// TwinCAT 3 PLC project Tc3EventLoggerUsage
// ProgramVersion: 3.1.4022.0
// libraries:
//   Tc2_MC2, * (Beckhoff Automation GmbH)
//   Tc2_Standard, * (Beckhoff Automation GmbH)
//   Tc2_System, * (Beckhoff Automation GmbH)
//   Tc2_Utilities, * (Beckhoff Automation GmbH)
//   Tc3_EventLogger, * (Beckhoff Automation GmbH)
//   Tc3_Module, * (Beckhoff Automation GmbH)
// project tree:
//   / GlobalTextList.TcGTLO, PlcTask.TcTTO, Visualization Manager.TcVMO (not stored), VISU_TASK.TcTTO
//   POUs/ FB_CONTROL.TcPOU, MAIN.TcPOU
//   VISUs/ Visualization.TcVIS
// (motion and I/O tree: see PLC project adslogeventexample)
// real-time tasks:
//   TASK PlcTask: cycle T#10ms, priority 20, ADS port 350
//   TASK VISU_TASK: cycle T#200000us, priority 30, ADS port 351
// variable links:
//   Tc3EventLoggerUsage/Tc3EventLoggerUsage Instance <-> NC-Task 1 SAF/Axes/Axis 1
//     PlcTask Inputs/MAIN.Axis.NcToPlc <-> Outputs/ToPlc
//     PlcTask Outputs/MAIN.Axis.PlcToNc <-> Inputs/FromPlc

CONFIGURATION Tc3EventLoggerUsage
    RESOURCE PLC ON TwinCAT3
        TASK PlcTask(INTERVAL := T#10ms, PRIORITY := 20);
        TASK VISU_TASK(INTERVAL := T#200000us, PRIORITY := 30);
        PROGRAM MAIN WITH PlcTask : MAIN;
        PROGRAM VisuElems_Visu_Prg WITH VISU_TASK : VisuElems.Visu_Prg;
    END_RESOURCE
END_CONFIGURATION

// ---- POUs/MAIN.TcPOU
PROGRAM MAIN
VAR
	control:fb_control;
	ServoPower:MC_Power;
	ServoReset:MC_Reset;
	Axis: AXIS_REF;
	Events:FB_AdsReadEvents;
	nNumberOfEvents: UDINT;
	bBusy: BOOL;
	bDone: BOOL;
	bError: BOOL;
	nErrId: UDINT;
END_VAR

control(Start:= control.Start, McOutputs=> , Axis:= Axis);

ServoPower(
	Axis:= Axis, 
	Enable:= ServoPower.Enable, 
	Enable_Positive:= TRUE, 
	Enable_Negative:= TRUE, 
	Override:= , 
	BufferMode:= MC_Aborting, 
	Options:= , 
	Status=> , 
	Busy=> , 
	Active=> , 
	Error=> , 
	ErrorID=> );

ServoReset(
	Axis:= Axis, 
	Execute:= ServoReset.Execute, 
	Done=> , 
	Busy=> , 
	Error=> , 
	ErrorID=> );	

	
Events(
	sNetId:= '', 
	bReadEvents:= Events.bReadEvents, 
	nLanguageId:= 1033, 
	eDateAndTimeFormat:= E_DateAndTimeFormat.de_DE, 
	tRefreshTime:= T#1S, 
	tTimeout:= T#5S, 
	aEvents=> , 
	nNumberOfEvents=> nNumberOfEvents, 
	bBusy=> bBusy, 
	bDone=> bDone, 
	bError=> bError, 
	nErrId=> nErrId);

END_PROGRAM

// ---- POUs/FB_CONTROL.TcPOU
FUNCTION_BLOCK FB_CONTROL
VAR_INPUT
	Start:BOOL;
END_VAR
VAR_OUTPUT
	McOutputs:ST_McOutputs;
END_VAR
VAR
	MoveAbsolute:MC_MoveAbsolute;
END_VAR

VAR_IN_OUT
	Axis: AXIS_REF;
END_VAR

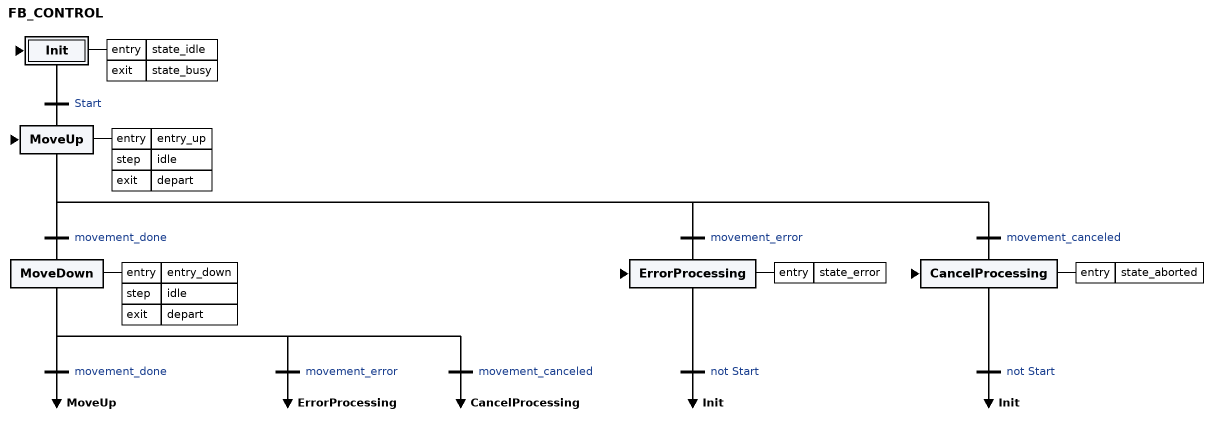
INITIAL_STEP Init:
    state_idle(P1);  // entry action
    state_busy(P0);  // exit action
END_STEP
TRANSITION FROM Init TO MoveUp
    := Start;
END_TRANSITION
STEP MoveUp:
    entry_up(P1);  // entry action
    idle(N);  // step action
    depart(P0);  // exit action
END_STEP
TRANSITION FROM MoveUp TO MoveDown
    := movement_done;
END_TRANSITION
TRANSITION FROM MoveUp TO ErrorProcessing
    := movement_error;
END_TRANSITION
STEP ErrorProcessing:
    state_error(P1);  // entry action
END_STEP
TRANSITION FROM ErrorProcessing TO Init
    := not Start;
END_TRANSITION
TRANSITION FROM MoveUp TO CancelProcessing
    := movement_canceled;
END_TRANSITION
STEP CancelProcessing:
    state_aborted(P1);  // entry action
END_STEP
TRANSITION FROM CancelProcessing TO Init
    := not Start;
END_TRANSITION
STEP MoveDown:
    entry_down(P1);  // entry action
    idle(N);  // step action
    depart(P0);  // exit action
END_STEP
TRANSITION FROM MoveDown TO MoveUp
    := movement_done;
END_TRANSITION
TRANSITION FROM MoveDown TO ErrorProcessing
    := movement_error;
END_TRANSITION
TRANSITION FROM MoveDown TO CancelProcessing
    := movement_canceled;
END_TRANSITION

ACTION depart:
MoveAbsolute.Execute:=FALSE;
idle();
END_ACTION

ACTION entry_down:
MoveAbsolute.Position:=0;
MoveAbsolute.Velocity:=100;
MoveAbsolute.Execute:=TRUE;
END_ACTION

ACTION entry_up:
MoveAbsolute.Position:=1000;
MoveAbsolute.Velocity:=100;
MoveAbsolute.Execute:=TRUE;
END_ACTION

ACTION idle:
MoveAbsolute(
	Axis:= Axis, 
	Execute:= , 
	Position:= , 
	Velocity:= , 
	Acceleration:= , 
	Deceleration:= , 
	Jerk:= , 
	BufferMode:= MC_Aborting, 
	Options:= , 
	Done=> , 
	Busy=> , 
	Active=> , 
	CommandAborted=> , 
	Error=> , 
	ErrorID=> );
END_ACTION

TRANSITION movement_canceled:
MoveAbsolute.CommandAborted;
END_TRANSITION

TRANSITION movement_done:
MoveAbsolute.Done;
END_TRANSITION

TRANSITION movement_error:
MoveAbsolute.Error;
END_TRANSITION

ACTION state_aborted:
McOutputs.CommandAborted:=TRUE;
McOutputs.Done:=
McOutputs.Busy:=
McOutputs.Active:=
McOutputs.Error:=FALSE;
McOutputs.ErrorID:=0;
END_ACTION

ACTION state_busy:
McOutputs.Busy:=TRUE;
McOutputs.Active:=
McOutputs.CommandAborted:=
McOutputs.Done:=
McOutputs.Error:=FALSE;
McOutputs.ErrorID:=0;
END_ACTION

ACTION state_done:
McOutputs.Busy:=
McOutputs.Active:=
McOutputs.CommandAborted:=
McOutputs.Done:=
McOutputs.Error:=FALSE;
McOutputs.ErrorID:=0;
END_ACTION

ACTION state_error:
McOutputs.Busy:=
McOutputs.Active:=
McOutputs.CommandAborted:=
McOutputs.Done:=FALSE;
McOutputs.Error:=TRUE;
McOutputs.ErrorID:=MoveAbsolute.ErrorID;
END_ACTION

ACTION state_idle:
McOutputs.Done:=TRUE;
McOutputs.Busy:=
McOutputs.Active:=
McOutputs.CommandAborted:=
McOutputs.Error:=FALSE;
McOutputs.ErrorID:=0;
END_ACTION

END_FUNCTION_BLOCK

// ---- GlobalTextList.TcGTLO
TEXTLIST GlobalTextList
  415 = 'Reset'
  721 = 'ServoOn'
  416 = 'Start'
END_TEXTLIST

// ---- VISUs/Visualization.TcVIS
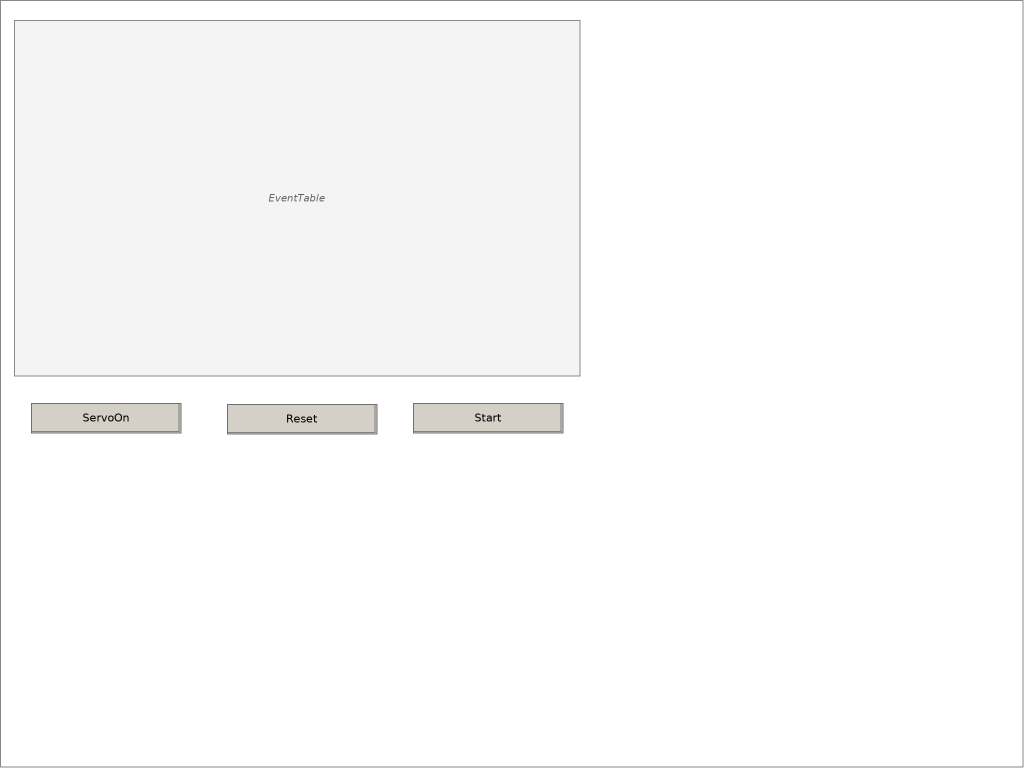
VISUALIZATION Visualization  // 1024x768
    EventTable (14,20 566x356)
        p1690906150: Class
        p3258520714: Date
        p2231227367: Time
        p3993844394: Message
        p2076579579: Details
        p3558512729: MAIN.Events.aEvents
        p3921149237: m_pDataArray..pArray
    Button (31,403 150x30), "ServoOn", pressed state: MAIN.ServoPower.Status
        toggle MAIN.ServoPower.Enable
    Button (413,403 150x30), "Start", pressed state: MAIN.control.McOutputs.Busy
        tap MAIN.control.Start
    Button (227,404 150x30), "Reset", pressed state: MAIN.ServoReset.Done
        tap MAIN.ServoReset.Execute
END_VISUALIZATION
